TYPE ST_SystemState :
STRUCT
	systemRUN: BOOL;
	systemSTOP: BOOL;
END_STRUCT
END_TYPE

(* stored: Version 1.1.0.1
   DUT ST_SystemState: Id {e6abef84-101c-43b8-b73d-9461b00ed4b4} *)
